FUNCTION_BLOCK OnLinkedListDisposedHandler EXTENDS OnLinkedListEventHandler

METHOD PUBLIC HandleEvent
VAR_INPUT
	Event : I_Event;
END_VAR
VAR
	linkedListDisposedEvent : I_LinkedListDisposedEvent;
END_VAR
IF __QUERYINTERFACE(Event, linkedListDisposedEvent) THEN
	_eventReceived := TRUE;
	fromExpected := linkedListDisposedEvent.TargetLinkedList = expectedOriginator;
END_IF
END_METHOD

END_FUNCTION_BLOCK

(* stored: Version 1.1.0.1, ProductVersion 3.1.4024.12
   POU OnLinkedListDisposedHandler: Id {b4a9c826-bbff-452b-b267-fe2dcde9cf76}, SpecialFunc None
   Method HandleEvent: Id {99fbacd1-95e1-45a9-b0ef-cd888ef75791} *)
